Xinje XDPPro project, PLC1: XD3-24 (software 3.7.5 2020-07-10)

PROGRAM Ladder

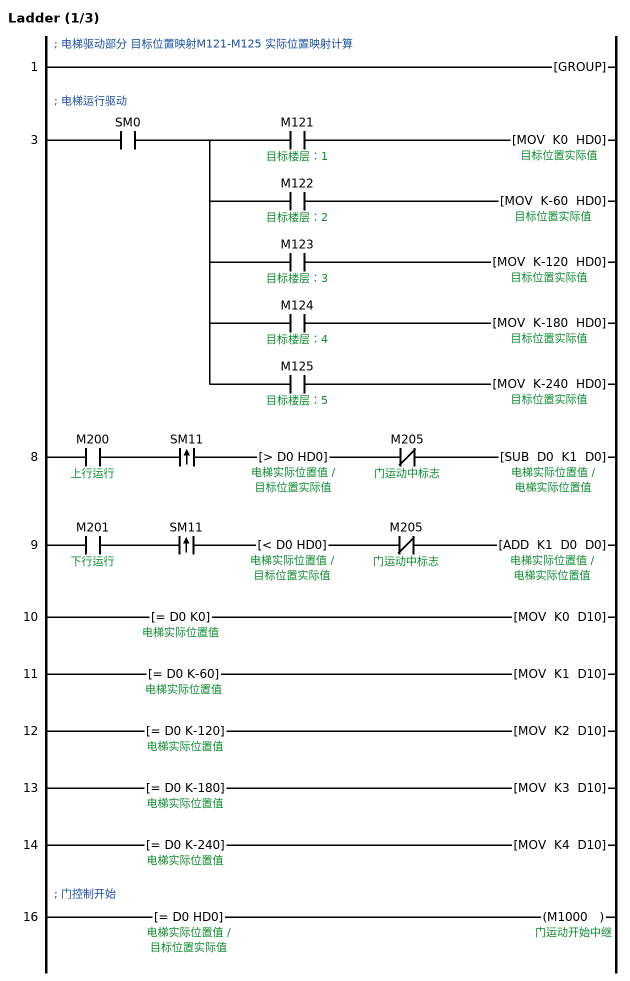
; 电梯驱动部分 目标位置映射M121-M125 实际位置映射计算
GROUP
; 电梯运行驱动
LD     SM0
MPS
AND    M121	; 目标楼层：1
MOV    K0 HD0	; 目标位置实际值
MRD
AND    M122	; 目标楼层：2
MOV    K-60 HD0	; 目标位置实际值
MRD
AND    M123	; 目标楼层：3
MOV    K-120 HD0	; 目标位置实际值
MRD
AND    M124	; 目标楼层：4
MOV    K-180 HD0	; 目标位置实际值
MPP
AND    M125	; 目标楼层：5
MOV    K-240 HD0	; 目标位置实际值
LD     M200	; 上行运行
ANDP   SM11
AND>   D0 HD0	; 电梯实际位置值 / 目标位置实际值
ANI    M205	; 门运动中标志
SUB    D0 K1 D0	; 电梯实际位置值 / 电梯实际位置值
LD     M201	; 下行运行
ANDP   SM11
AND<   D0 HD0	; 电梯实际位置值 / 目标位置实际值
ANI    M205	; 门运动中标志
ADD    K1 D0 D0	; 电梯实际位置值 / 电梯实际位置值
LD=    D0 K0	; 电梯实际位置值
MOV    K0 D10
LD=    D0 K-60	; 电梯实际位置值
MOV    K1 D10
LD=    D0 K-120	; 电梯实际位置值
MOV    K2 D10
LD=    D0 K-180	; 电梯实际位置值
MOV    K3 D10
LD=    D0 K-240	; 电梯实际位置值
MOV    K4 D10
; 门控制开始
LD=    D0 HD0	; 电梯实际位置值 / 目标位置实际值
OUT    M1000	; 门运动开始中继

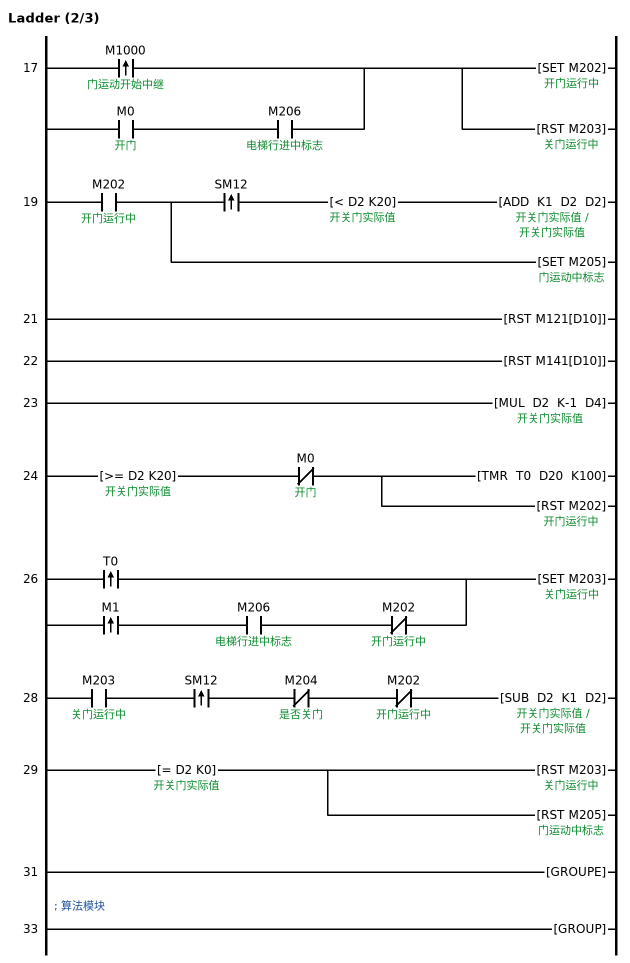
LDP    M1000	; 门运动开始中继
LD     M0	; 开门
AND    M206	; 电梯行进中标志
ORB
SET    M202	; 开门运行中
RST    M203	; 关门运行中
LD     M202	; 开门运行中
MPS
ANDP   SM12
AND<   D2 K20	; 开关门实际值
ADD    K1 D2 D2	; 开关门实际值 / 开关门实际值
MPP
SET    M205	; 门运动中标志
RST    M121[D10]
RST    M141[D10]
MUL    D2 K-1 D4	; 开关门实际值
LD>=   D2 K20	; 开关门实际值
ANI    M0	; 开门
TMR    T0 D20 K100
RST    M202	; 开门运行中
LDP    T0
LDP    M1
AND    M206	; 电梯行进中标志
ANI    M202	; 开门运行中
ORB
SET    M203	; 关门运行中
LD     M203	; 关门运行中
ANDP   SM12
ANI    M204	; 是否关门
ANI    M202	; 开门运行中
SUB    D2 K1 D2	; 开关门实际值 / 开关门实际值
LD=    D2 K0	; 开关门实际值
RST    M203	; 关门运行中
RST    M205	; 门运动中标志
GROUPE
; 算法模块
GROUP

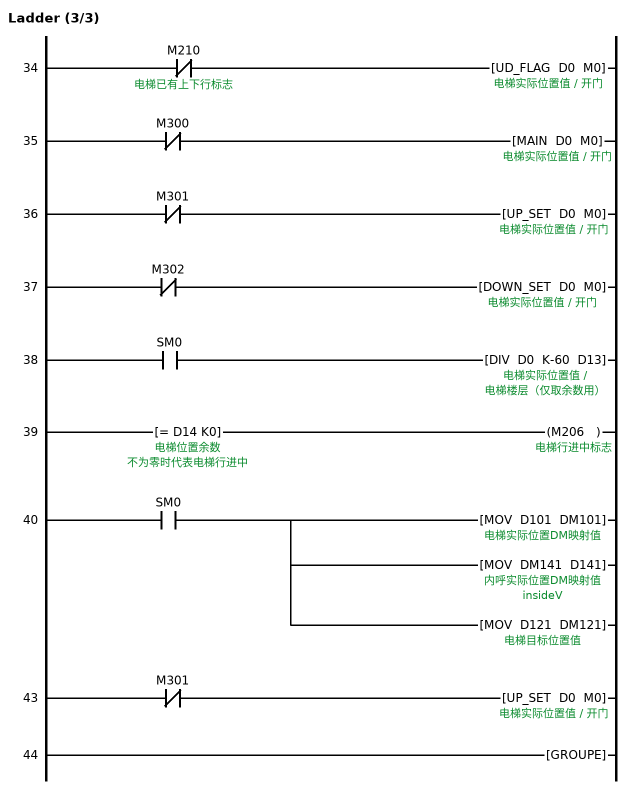
LDI    M210	; 电梯已有上下行标志
UD_FLAG D0 M0	; 电梯实际位置值 / 开门
LDI    M300
MAIN   D0 M0	; 电梯实际位置值 / 开门
LDI    M301
UP_SET D0 M0	; 电梯实际位置值 / 开门
LDI    M302
DOWN_SET D0 M0	; 电梯实际位置值 / 开门
LD     SM0
DIV    D0 K-60 D13	; 电梯实际位置值 / 电梯楼层（仅取余数用）
LD=    D14 K0	; 电梯位置余数 不为零时代表电梯行进中
OUT    M206	; 电梯行进中标志
LD     SM0
MOV    D101 DM101	; 电梯实际位置DM映射值
MOV    DM141 D141	; 内呼实际位置DM映射值 insideV
MOV    D121 DM121	; 电梯目标位置值
LDI    M301
UP_SET D0 M0	; 电梯实际位置值 / 开门
GROUPE

COMMENTS (devices not used above)
D58	dv_up
D57	P
D56	a
D59	ins
D60	c
D61	d
M141	内呼位映射 inside
M101	电梯实际位置位映射
D62	up_down_dif

C FUNCTION BLOCK down_set.fcb
/*************************************************************************
   FunctionBlockName:  DOWN_SET
   Version:            1.0.0
   Author:             
   UpdateTime:         2020/8/31 16:01:39
   Comment:            
			
**************************************************************************/
 
#include"define.h"
 


void DOWN_SET( WORD W , BIT B )
{
//#define SysRegAddr_HD_D_HM_M
    int F,s,v,i;

    buf[factP]=0;//清除内呼楼层分离储存数组对应元素
    v=0;
    for(i=0;i<factP;i++)
    {   
        v=v+buf[i];

}
    if(v==0)
{
        B[201]=0;
}
    //DOWN_SET主程序开始
    if(B[200]==0&&B[201]==0){
        targetV=0;
        }
    if(B[201]==1){
        
        B[302]=1;
        F=factP;
        //targetV=buf[F];
    while(F>=0)
        {//s=buf[F];
            if(buf[F]!=0){
                    targetV=buf[F];
                    break;
                       // F=D[80];
                    }
            if(buf[F]==0){
                    F=F-1;
                    }
    }
    B[302]=0;
    }


}

C FUNCTION BLOCK first.fcb
/*************************************************************************
   FunctionBlockName:  FIRST
   Version:            1.0.0
   Author:             rosireity
   UpdateTime:         2020/9/12 8:43:36
   Comment:            
			
**************************************************************************/


#include "define.h" 


void FIRST( WORD W , BIT B )
{
 

}

C FILE define.h
#ifndef	_DEFINE_H
#define	_DEFINE_H
#include"SYS.h"
#define factV           D[101]      //电梯实际位置（整数滞后） 数值
#define targetV        D[121]      //电梯目标位置 数值
#define factP           D[10]       //电梯实际位置 楼层
#define remainderP    D[14]       //电梯实际位置余数 用于确定是否在楼层间
#define insideV         D[141]      //电梯内呼位置 数值
#define P                 D[12]       //factP+1  
int buf[5];                              //内呼楼层分离储存数组
#endif

C FILE pow.h
#ifndef	_POW_H
#define	_POW_H
#endif


/***********次方***********/
int pow(a,b)
{
    int a,b,c,i;
    c=a;
    if(b==0)
    {
        return 1;
        }
    for(i=0;i<b;i++)
    {
        
        c=c*a;
        }
     return c;
}

C FILE sys.h
#ifndef OVERRIDE
	#define OVERRIDE
#endif
//2019.11.25
//V1.0.0

#ifdef ARM_M3M4
typedef INT32U ARM_BIT;
#else
typedef INT8U ARM_BIT;
#endif

#ifndef HEAD_SYS_REG_ADDR

#define HEAD_SYS_REG_ADDR

#define SYSREGADDR_VISION_2

#pragma region SysRegAddr

    //引用类型
    extern char  __X;
	extern char  __Y;
    extern char  __M;
    extern char  __SM;
	extern char  __HM;
	extern char  __T;
	
	extern short __D;
	extern short __HD;
	extern short __SD;
	extern short __HSD;
	extern short __HSCD;
	extern short __FD;
	extern short __SFD;
	extern short __SSFD;
	extern short __ID;
	extern short __QD;
	extern short __CD;

	

    
	#define D			(&__D)
	#define CD			(&__CD)
	#define HD			(&__HD)
	#define SD			(&__SD)
	#define HSD		(&__HSD)
	#define HSCD		(&__HSCD)
	#define FD			(&__FD)
	#define SFD		(&__SFD)
	#define SSFD		(&__SSFD)
	#define ID			(&__ID)
	#define QD			(&__QD)

	#define M_			((ARM_BIT *)(&__M))
	#define HM_		((ARM_BIT *)(&__HM))
	#define SM_		((ARM_BIT *)(&__SM))
	#define X_			((ARM_BIT *)(&__X))
	#define Y_			((ARM_BIT *)(&__Y))

	#define DHSCD		*(INT32S *)&HSCD
	#define DHSD		*(INT32S *)&HSD
	#define LHSD		*(long long *)&HSD
	#define DSD			*(INT32S *)&SD
	#define FSD			*(FP32 *)&SD
	#define LSD			*(long long *)&SD
	#define DHD			*(INT32S *)&HD
	#define FHD			*(FP32 *)&HD
	#define LHD			*(long long *)&HD
	#define DFD			*(INT32S *)&FD
	#define FFD			*(FP32 *)&FD
	#define DD			*(INT32S *)&D
	#define LDD			*(long long *)&D
	#define FDD			*(FP32 *)&D
	#define DW			*(INT32S*)&W
	#define FW      	*(FP32*)&W
	#define LW      	*(long long *)&W
	#define DID			*(INT32S *)&ID
	#define DQD			*(INT32S *)&QD
    #define DSFD		*(INT32S *)&SFD
    #define FSFD		*(FP32 *)&SFD
    #define LSFD		*(long long *)&SFD
#pragma endregion


#endif

C FUNCTION BLOCK main.fcb
/*************************************************************************
   FunctionBlockName:  MAIN
   Version:            1.0.0
   Author:             rosireity
   UpdateTime:         2020/8/31 16:01:39
   Comment:            
			
**************************************************************************/    


#include "define.h" 

       
void MAIN( WORD W , BIT B )
{   
    //0#define SysRegAddr_HD_D_HM_M
    
    int a,b,c,d,e,f,g,h,i,j,k,l,m,n,F;
    //buf[5]={0};
    int dv_up,dv_down,ins;
    

    /*********************M映射**********************/
    

    factV = pow(2,(int)factP);  //实际楼层位置DM
    P=factP+1;
    D[57]=P;
 
    /*********************上下行分配标志获取**********************/
    
    
    if(B[200]==1||B[201]==1)
    {
        B[210]=1;
        }
    else
    {
        B[210]=0;
        }
    

    /*********************内呼处理**********************/
    

        
        dv_up=5;
        D[58]=dv_up;
        f=insideV;
        c=4;
        B[300]=1;//切除MAIN函数重复运行
        while(dv_up>0)
        {
        
        d=pow(2,c);
        //D[61]=d;
        ins=f-d;
        //D[59]=ins;
        
        if(ins>=0)
        {
                //a=dv_up;
                buf[c]=pow(2,c);
                dv_up=dv_up-1;
                f=f-d;
                //D[56]=a;
                c=c-1;
                //D[60]=c;
                //if(c==P)
                //{break;}
            
        }
            else
            {
                dv_up=dv_up-1;
                buf[c]=0;
                c=c-1;
            
            }
        //数据分离结束
        
        //清除上行标志位
        //e=factP+1;
        
        //targetV=buf[P];
        B[300]=0; //MAIN函数重新运行   
                
}//上行处理结束

        D[55]=buf[4];
        D[54]=buf[3];
        D[53]=buf[2];
        D[52]=buf[1];
        D[51]=buf[0];
                
}

C FUNCTION BLOCK ud_flag.fcb
/*************************************************************************
   FunctionBlockName:  UD_FLAG
   Version:            1.0.0
   Author:             
   UpdateTime:         2020/8/31 18:07:45
   Comment:            
			
**************************************************************************/


#include "define.h"

 
void UD_FLAG( WORD W , BIT B )
{
    
    //#define SysRegAddr_HD_D_HM_M     
    int up_down_dif;
    

    /*********************M映射**********************/
    

    factV = pow(2,(int)factP);  //实际楼层位置
    
    
    /*********************上下行标志获取**********************/
    
    up_down_dif=(int)insideV-(int)factV;
    D[62]=up_down_dif;

    
    if(insideV!=0&&up_down_dif>0)
    {
        B[200]=1;
        }
    if(insideV!=0&&up_down_dif<0)
    {
        B[201]=1;
        }
    if(insideV==0&&remainderP==0)
    {
        B[200]=0;
        B[201]=0;
        }


}

C FUNCTION BLOCK up_set.fcb
/*************************************************************************
   FunctionBlockName:  UP_SET
   Version:            1.0.0
   Author:             rosireity
   UpdateTime:         2020/8/31 16:01:39
   Comment:            
			
**************************************************************************/
 
#include"define.h"


void UP_SET( WORD W , BIT B )
{
    
    int F,s,v,i;
    
    buf[factP]=0;//清除内呼楼层分离储存数组对应元素
    v=0;
    for(i=4;i>=factP;i--)
    {   
        v=v+buf[i];
        //D[64]=v;
        //D[65]=i;
}
    if(v==0)
{
        B[200]=0;
}
    //UP_SET主程序开始
    if(B[200]==0&&B[201]==0){
        targetV=0;
        }
    if(B[200]==1){
        
        B[301]=1;
        F=factP;
        //targetV=buf[F];
    while(F<5)
        {//s=buf[F];
            if(buf[F]!=0){
                    targetV=buf[F];
                    break;
                       // F=D[80];
                    }
            if(buf[F]==0){
                    F=F+1;
                    }
    }
    B[301]=0;
    }
    
    

}